FUNCTION_BLOCK Comparator (* Composite Function Block Type *)
  (* Standard: 61499-2 *)
  (* Version 0.0, 12/10/2023, Cheyan, Schneider Electric, template *)
  PACKAGE Main;
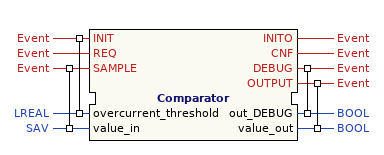
  EVENT_INPUT
    INIT WITH overcurrent_threshold; (* Initialization Request *)
    REQ; (* Normal Execution Request *)
    SAMPLE WITH value_in;
  END_EVENT
  EVENT_OUTPUT
    INITO; (* Initialization Confirm *)
    CNF; (* Execution Confirmation *)
    DEBUG WITH out_DEBUG;
    OUTPUT WITH value_out;
  END_EVENT
  VAR_INPUT
    overcurrent_threshold : LREAL;
    value_in : SAV; (* Input event qualifier *)
  END_VAR
  VAR_OUTPUT
    out_DEBUG : BOOL;
    value_out : BOOL;
  END_VAR
  (* Comparator Comment *)
  FBS
    FB1 : PIOC_Logic;
  END_FBS
  EVENT_CONNECTIONS
    INIT TO FB1.INIT;
    REQ TO FB1.REQ;
    FB1.INITO TO INITO;
    FB1.CNF TO CNF;
    FB1.DEBUG TO DEBUG;
    SAMPLE TO FB1.SAMPLE;
    FB1.OUTPUT TO OUTPUT;
  END_CONNECTIONS
  DATA_CONNECTIONS
    overcurrent_threshold TO FB1.overcurrent_threshold;
    FB1.out_DEBUG TO out_DEBUG;
    value_in TO FB1.in_value;
    FB1.out_value TO value_out;
  END_CONNECTIONS
END_FUNCTION_BLOCK
